(*			
	RafalOS
	Rafał Osajda		20.11.2025		TC 4024.66
	Moduł przygotowania danych dla Okna ustawień we wszystkich trybach
*)
FUNCTION_BLOCK FB_MCHMIPrepareDataForScreen_07_XX EXTENDS FB_MCHMIPrepareDataForScreen IMPLEMENTS ITF_MCHMIPrepareDataForScreen
VAR
	itfMachineControlHMI	: ITF_MCHMIMachineControl_HMI_PrepScr_07_XX;
	refstData				: REFERENCE TO ST_MCHMIPrepareScreen_07_XX;
END_VAR

(*			
	RafalOS
	Rafał Osajda		19.11.2025		TC 4024.66
	Czyści danych przy zmienia ramki po poprzedniej ramce
*)
METHOD PUBLIC ClearAfterScreen : BOOL
VAR_INPUT
END_VAR
SUPER^.ClearAfterScreen ();
END_METHOD

METHOD PUBLIC LinkDataHMI_07_XX : BOOL
VAR_INPUT
	refstData				: REFERENCE TO ST_MCHMIPrepareScreen_07_XX;
END_VAR
THIS^.refstData REF= refstData;
END_METHOD

METHOD PUBLIC LinkMachineControlHMI : BOOL
VAR_INPUT
	fbMachineControlHMI	: ITF_MCHMIMachineControl_HMI_PrepScr_07_XX;
END_VAR
this^.itfMachineControlHMI := fbMachineControlHMI;
END_METHOD

(*			
	RafalOS
	Rafał Osajda		14.11.2025		TC 4024.66
	Metoda przygotowywania danych dla HMI 
	W niej odbywa się odpytywanie właściego elementu przez łącznik
*)
METHOD PUBLIC PrepareDataForHMI : BOOL
VAR_INPUT
END_VAR
	(*	Zmiana języka - przygotowanie listy dostępnych języków	*)
THIS^.SettingLocation ();
	
IF (THIS^.refstData.bCreateRecipeTemplate) THEN
	THIS^.refstData.bCreateRecipeTemplate := FALSE;
	THIS^.itfMachineControlHMI.CreateRecipeTemplates ();
END_IF

	(*	Rozszerzenie wyświetlania	*)
SUPER^.PrepareDataForHMI ();
END_METHOD

(*			
	RafalOS
	Rafał Osajda		19.11.2025		TC 4024.66
	Przygotowanie ramki pood tamke do wyświetlenia - tylko przygotowanie a nie przygotowanie danych do wyświetlenia
*)
METHOD PUBLIC PrepareForScreen : BOOL
VAR_INPUT
END_VAR
SUPER^.PrepareForScreen ();
END_METHOD

METHOD PRIVATE SettingLocation : BOOL
VAR_INPUT
END_VAR

VAR
	iI: INT;
	sCodeLocation: STRING;
END_VAR
IF (THIS^.refstHMICommonData.bChangePage) THEN
	FOR iI := 1 TO GVL_BaseConstans.NUMBER_OF_LOCATIONS DO
		THIS^.refstData.arrLocationDescription [iI-1] := THIS^.refstCommonData.itfLocaciotn.GetDescription (iIN := iI);
	END_FOR
	THIS^.refstData.iChoosoLocation := TO_INT (THIS^.refstCommonData.itfLocaciotn.GetLocation ()) - 1;
END_IF

IF ((THIS^.refstData.iChoosoLocation + 1) <> TO_INT (THIS^.refstCommonData.itfLocaciotn.GetLocation ())) THEN
	sCodeLocation := TO_STRING (THIS^.refstCommonData.itfLocaciotn.GetCode (iIN := THIS^.refstData.iChoosoLocation + 1));
	THIS^.refstCommonData.itfLocaciotn.SetLocation (sLocation := TO_STRING (sCodeLocation));
	CURRENTLANGUAGE := sCodeLocation;
END_IF

(*

IF (THIS^.refstOHMI.stUstawienia.iWybranyJezyk <> (TO_INT (THIS^.fbLokalizacja.getJezyk ()) - 1)) THEN
	THIS^.fbLokalizacja.setJezyk (sNowy				:= THIS^.fbLokalizacja.zwrocKod (iIN := THIS^.refstOHMI.stUstawienia.iWybranyJezyk + 1));
	VisuElems.CURRENTLANGUAGE							:= THIS^.fbLokalizacja.zwrocAktualnyKod ();
END_IF
*)
END_METHOD

END_FUNCTION_BLOCK

(* stored: Version 1.1.0.1
   POU FB_MCHMIPrepareDataForScreen_07_XX: Id {7d8c545d-4c9d-09fa-250b-a18c25f3ac38}, SpecialFunc None
   Folder ITF_PDFS: Id {15561f8c-f596-0f6c-0f44-98a5c11de2d4}
   Method ClearAfterScreen: Id {fce75c41-804a-01d1-00bf-14670fe683ea}
   Method LinkDataHMI_07_XX: Id {170edd4d-76e4-01f2-04ab-358ca7c84492}
   Method LinkMachineControlHMI: Id {03329350-272a-02cd-1ccc-806af2e0c0f0}
   Method PrepareDataForHMI: Id {5852a739-6009-0e53-3110-3d91ee9d862e}
   Method PrepareForScreen: Id {0cacd757-89e8-0ff8-1488-6cd1abe331a7}
   Method SettingLocation: Id {fcbc6cbc-e79a-0bba-2afe-192439bfcb6a} *)
